Yaskawa INFORM job: R1_W30(0,0)OK-KM.JBI

/JOB
//NAME R1_W30(0,0)OK-KM
///FOLDERNAME KRIS-SCIANA
//POS
///NPOS 58,58,0,5,0,0
///TOOL 0
///POSTYPE PULSE
///PULSE
C00000=7475,65197,-10516,-9470,81833,84687
C00001=-14781,-136725,-123062,2478,40093,78051
C00002=-47735,-136725,-131238,2478,40093,78051
C00003=-106770,-122317,-131129,58923,70663,56463
C00004=-139981,-114211,-111146,90677,87861,44317
C00005=-139981,-114211,-111146,90677,87861,44317
C00006=-75386,-3535,-30317,66464,85013,44761
C00007=-66538,11642,-20496,54302,72109,39274
C00008=-65112,17030,-10985,54607,69462,38360
C00009=-64572,18263,-9841,54433,69113,38445
C00010=-65112,17030,-10985,54607,69462,38360
C00011=-65112,16871,-10085,54794,69084,38109
C00012=-65112,17030,-10985,54607,69462,38360
C00013=-63397,8717,-18491,53875,68708,38853
C00014=-63017,11492,-11966,54556,66933,37907
C00015=-62693,12252,-11285,54447,66730,37964
C00016=-63017,11492,-11966,54556,66933,37907
C00017=-63383,13303,-10334,54708,67099,37801
C00018=-63017,11492,-11966,54556,66933,37907
C00019=-55759,-6604,-27311,51741,62959,39574
C00020=-55661,-6462,-27483,51631,63020,39665
C00021=-55185,-5230,-26493,51425,62774,39784
C00022=-55661,-6462,-27483,51631,63020,39665
C00023=-54802,-7286,-28141,51284,62538,39860
C00024=-55661,-6462,-27483,51631,63020,39665
C00025=-55661,-5963,-30702,50797,64457,40544
C00026=-51909,-5737,-34456,44523,67327,43326
C00027=-51589,-4824,-33719,44375,67186,43412
C00028=-51909,-5737,-34456,44523,67327,43326
C00029=-51909,-5927,-33812,44665,66970,43155
C00030=-51909,-5737,-34456,44523,67327,43326
C00031=-54286,-11411,-41702,45169,69574,43269
C00032=-50718,587,-32012,42945,73869,38021
C00033=-51522,1958,-30394,43322,74026,37730
C00034=-53169,4824,-27534,44022,74582,37240
C00035=-53820,5829,-26500,44295,74806,37046
C00036=-55870,1186,-31537,44958,76292,36795
C00037=-59392,9299,-24533,46716,78497,-24031
C00038=-63863,20602,2697,63471,79674,-34385
C00039=-63934,21237,8063,63937,78335,-35635
C00040=-65732,24427,4489,63688,81267,-34323
C00041=-46082,-27287,-40473,14267,37051,-7026
C00042=-46140,-18492,-30342,14917,35402,-7384
C00043=-45824,-18838,-28527,15037,34090,-7469
C00044=-45694,-18742,-25675,15567,32416,-7759
C00045=-45367,-24360,-34633,14175,34900,-7028
C00046=-40689,-6131,-37024,-1176,62534,-55068
C00047=-47219,-13016,-42982,8463,53187,-56644
C00048=-54487,10408,-27704,19037,64046,-63382
C00049=-55342,15666,-21575,22074,65650,-65542
C00050=-52751,10069,-25477,20680,64583,-64792
C00051=-53093,2120,-32761,20812,65035,-64831
C00052=-68304,-26780,-65179,28219,73809,-68361
C00053=-139981,-114211,-111146,90677,87861,44317
C00054=-139981,-114211,-111146,90677,87861,44317
C00055=-139981,-161315,-135562,90677,60865,44317
C00056=-139981,-161315,-135562,90677,60865,44317
C00057=-32105,35387,-19670,23246,82833,71797
BC00000=161490,337827,1074007
BC00001=326897,13670,1070569
BC00002=34574,13670,1070569
BC00003=12457,4931,1066314
BC00004=15,15,1063921
BC00005=15,15,176683
BC00006=15,15,182318
BC00007=15,4078,182318
BC00008=15,4078,182318
BC00009=15,4078,182318
BC00010=15,4078,182318
BC00011=15,4078,182318
BC00012=15,4078,182318
BC00013=15,4078,182318
BC00014=15,4078,182318
BC00015=15,4078,182318
BC00016=15,4078,182318
BC00017=15,4078,182318
BC00018=15,4078,182318
BC00019=15,4078,182318
BC00020=15,4078,182318
BC00021=15,4078,182318
BC00022=15,4078,182318
BC00023=15,4078,182318
BC00024=15,4078,182318
BC00025=15,4078,182318
BC00026=15,4078,182318
BC00027=15,4078,182318
BC00028=15,4078,182318
BC00029=15,4078,182318
BC00030=15,4078,182318
BC00031=15,4078,182318
BC00032=15,4078,182318
BC00033=15,4078,182318
BC00034=15,4078,182318
BC00035=15,4078,182316
BC00036=15,4078,182316
BC00037=15,4078,182314
BC00038=15,4078,182314
BC00039=15,4078,182314
BC00040=15,4078,182314
BC00041=15,4078,182314
BC00042=15,4078,182314
BC00043=15,4078,182314
BC00044=15,4078,182314
BC00045=15,4078,182314
BC00046=15,4078,182314
BC00047=15,4078,182314
BC00048=15,4078,182313
BC00049=15,4078,182312
BC00050=15,4078,182312
BC00051=15,4078,182312
BC00052=15,4078,182312
BC00053=15,15,176683
BC00054=15,15,1063921
BC00055=15,15,1063921
BC00056=364339,15,1063921
BC00057=200004,395,1071100
///POSTYPE BASE
///RECTAN
///RCONF 0,0,0,0,1,0,0,0,0,0,0,0,0,0,0,0,0,0,0,0,0,0,0,0
P00006=2.006,1.622,-0.565,0.0000,0.0000,0.0000
P00022=2.006,1.622,-0.565,0.0000,0.0000,0.0000
///RCONF 0,0,0,0,0,0,0,0,0,0,0,0,0,0,0,0,0,0,0,0,0,0,0,0
P00023=-2.957,-4.083,2.762,0.0000,0.0000,0.0000
P00024=-1.466,-0.226,-0.419,0.0000,0.0000,0.0000
P00025=3.643,0.007,-2.585,0.0000,0.0000,0.0000
//INST
///DATE 2024/09/16 12:05
///ATTR SC,RW
///GROUP1 RB1,BS1
NOP
'r1_W30(0,0)
'Path VIA1137
SFTOF
MOVJ C00000 BC00000 VJ=100.00
MOVJ C00001 BC00001 VJ=50.00
MOVJ C00002 BC00002 VJ=100.00
MOVJ C00003 BC00003 VJ=100.00
MOVJ C00004 BC00004 VJ=100.00
'BRAK BLASZEK
MOVJ C00005 BC00005 VJ=100.00
MOVJ C00006 BC00006 VJ=50.00
MOVJ C00007 BC00007 VJ=50.00
MOVJ C00008 BC00008 VJ=15.00
REFP 3 C00009 BC00009
CALL JOB:SEARCH-R1
SET P022 P006
SFTON P022
MOVL C00010 BC00010 V=60.0
REFP 3 C00011 BC00011
CALL JOB:SEARCH-R1
SET P022 P006
SFTON P022
MOVL C00012 BC00012 V=60.0
MOVL C00013 BC00013 V=100.0
MOVL C00014 BC00014 V=100.0
REFP 3 C00015 BC00015
CALL JOB:SEARCH-R1
SET P023 P006
SFTON P023
MOVL C00016 BC00016 V=60.0
REFP 3 C00017 BC00017
CALL JOB:SEARCH-R1
SET P023 P006
SFTON P023
MOVL C00018 BC00018 V=60.0
MOVL C00019 BC00019 V=100.0
MOVL C00020 BC00020 V=100.0
REFP 3 C00021 BC00021
CALL JOB:SEARCH-R1
SET P025 P006
SFTON P025
MOVL C00022 BC00022 V=60.0
REFP 3 C00023 BC00023
CALL JOB:SEARCH-R1
SET P025 P006
SFTON P025
MOVL C00024 BC00024 V=60.0
MOVL C00025 BC00025 V=100.0
MOVL C00026 BC00026 V=100.0
REFP 3 C00027 BC00027
CALL JOB:SEARCH-R1
SET P024 P006
SFTON P024
MOVL C00028 BC00028 V=60.0
REFP 3 C00029 BC00029
CALL JOB:SEARCH-R1
SET P024 P006
SFTON P024
MOVL C00030 BC00030 V=60.0
MOVL C00031 BC00031 V=100.0
CALL JOB:COFNIJ_DRUT
MACRO1 MJ#(0) ARGF7
SFTON P024
MOVL C00032 BC00032 V=100.0
ARCON
MOVL C00033 BC00033 V=10.0
MOVL C00034 BC00034 V=10.0
MOVL C00035 BC00035 V=10.0
ARCOF
MOVJ C00036 BC00036 VJ=15.00
SFTOF
MOVJ C00037 BC00037 VJ=15.00
SFTON P025
MOVL C00038 BC00038 V=83.3
ARCON
MOVL C00039 BC00039 V=11.7
ARCOF
MOVL C00040 BC00040 V=83.3
SFTOF
MOVL C00041 BC00041 V=83.3
SFTON P023
MOVL C00042 BC00042 V=83.3
ARCON
MOVL C00043 BC00043 V=11.7
MOVL C00044 BC00044 V=11.7
ARCOF
MOVJ C00045 BC00045 VJ=15.00
SFTOF
MOVJ C00046 BC00046 VJ=20.00
MOVJ C00047 BC00047 VJ=20.00
MOVJ C00048 BC00048 VJ=40.00
SFTON P022
MOVJ C00049 BC00049 VJ=20.00
ARCON
MOVL C00050 BC00050 V=10.0
ARCOF
MOVJ C00051 BC00051 VJ=20.00
SFTOF
MOVJ C00052 BC00052 VJ=40.00
MOVJ C00053 BC00053 VJ=40.00
MOVJ C00054 BC00054 VJ=100.00
MOVJ C00055 BC00055 VJ=70.00
MOVJ C00056 BC00056 VJ=100.00
MOVJ C00057 BC00057 VJ=100.00
END
